// TIA Portal V17 export
// export: Created 2023-12-22T15:08:07.2118922Z, ExportSetting WithDefaults, DisplayName Totally Integrated Automation Portal, DisplayVersion V17, DisplayName TIA Portal Openness, DisplayVersion V17, DisplayName TIA Portal Version Control Interface, DisplayVersion V17, DisplayName STEP 7 Professional, DisplayVersion V17, DisplayName STEP 7 Safety, DisplayVersion V17, DisplayName WinCC Advanced, DisplayVersion V17
FUNCTION_BLOCK "Time_S_b"   // FB89, LAD
{ S7_Optimized_Access := 'FALSE' }
VERSION : 0.1
// stored: AutoNumber false, IsIECCheckEnabled false, SetENOAutomatically false, UDAEnableTagReadback false
   VAR DB_SPECIFIC
      SP { S7_SetPoint := 'True'} : Byte := 2;   // Уставка
      Now : Byte;   // Текущий счёт
      Start : Bool;   // Запуск
      "Exit" : Bool;   // Счёт завершён
      Pause : Bool;   // Пауза
      Reset : Bool;   // Сброс таймера
   END_VAR
   VAR_TEMP   // added for the SCL form of the ladder/FBD networks
      _w1 : Bool;
   END_VAR
BEGIN

REGION Network 1: Подсчёт времени
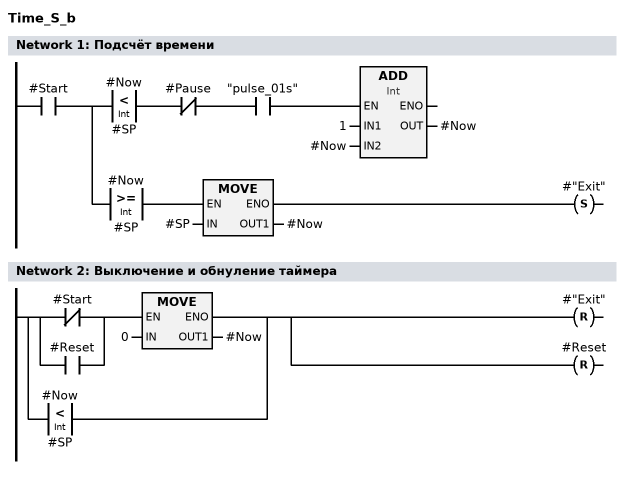
   RUNG wire#powerrail
      Contact( #Start )
      wire#w1
      { S7_Templates := "SrcType := Int" } LT_Contact(in1 := #Now, in2 := #SP)
      I_Contact( #Pause )
      Contact( "pulse_01s" )
      { S7_Templates := "SrcType := Int"; S7_GenerateENO := "TRUE" } Add(in1 := 1, in2 := #Now, out => #Now)
   END_RUNG
   RUNG wire#w1
      { S7_Templates := "SrcType := Int" } GE_Contact(in1 := #Now, in2 := #SP)
      { S7_GenerateENO := "TRUE" } Move(in := #SP, out1 => #Now)
      S_Coil( #"Exit" )
   END_RUNG
   // the same network as SCL:
   // ENO of a box is taken as its EN; it also drops when the box reports an error
   IF #Start AND (#Now < #SP) AND NOT #Pause AND "pulse_01s" THEN #Now := 1 + #Now; END_IF;
   #_w1 := #Start AND (#Now >= #SP);
   IF #_w1 THEN
       #Now := #SP;
       #"Exit" := TRUE;
   END_IF;
END_REGION

REGION Network 2: Выключение и обнуление таймера
   RUNG wire#powerrail
      I_Contact( #Start )
      wire#w1
      { S7_GenerateENO := "TRUE" } Move(in := 0, out1 => #Now)
      wire#w2
      R_Coil( #"Exit" )
   END_RUNG
   RUNG wire#powerrail
      Contact( #Reset )
   END_RUNG wire#w1
   RUNG wire#powerrail
      { S7_Templates := "SrcType := Int" } LT_Contact(in1 := #Now, in2 := #SP)
   END_RUNG wire#w2
   RUNG wire#w2
      R_Coil( #Reset )
   END_RUNG
   // the same network as SCL:
   // ENO of a box is taken as its EN; it also drops when the box reports an error
   #_w1 := NOT #Start OR #Reset;
   IF #_w1 THEN #Now := 0; END_IF;
   IF #_w1 OR (#Now < #SP) THEN
       #"Exit" := FALSE;
       #Reset := FALSE;
   END_IF;
END_REGION
END_FUNCTION_BLOCK
